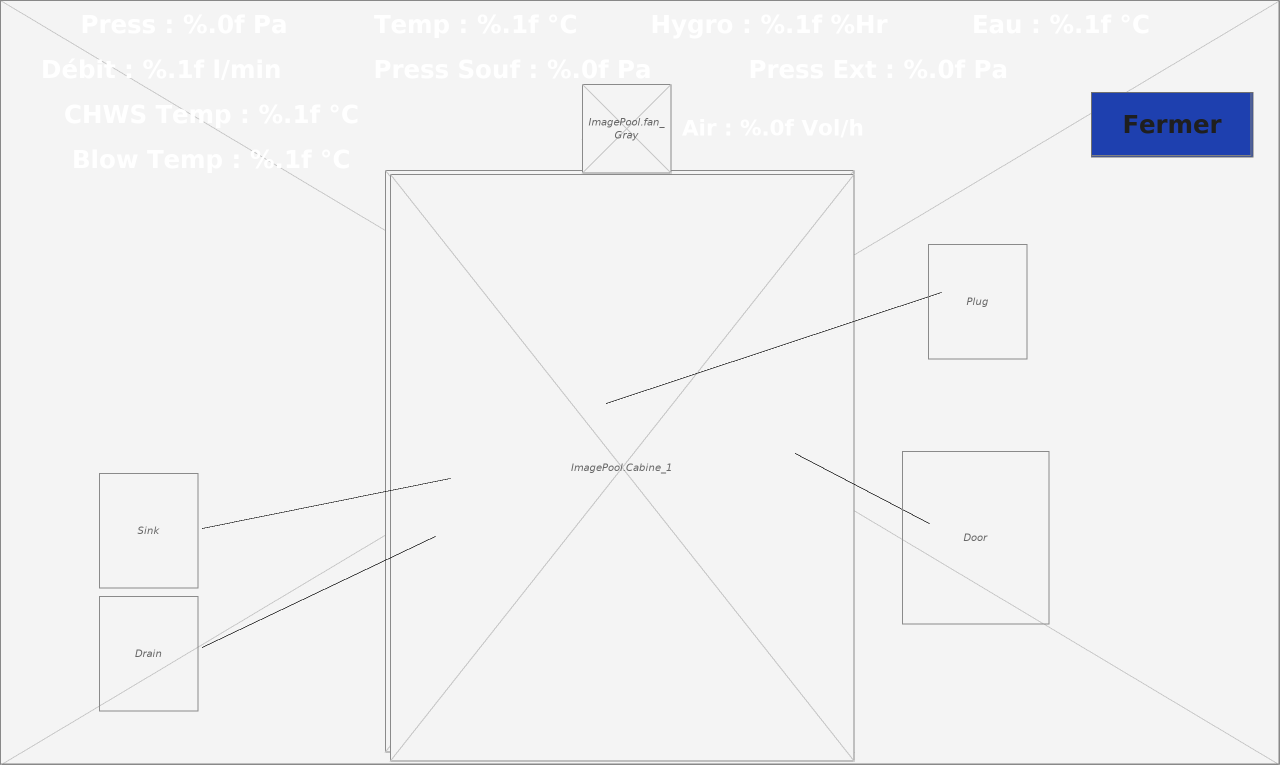
VISUALIZATION Actionneurs  // 1280x765
    Image (0,0 1280x765), image: ImagePool.Fond_Degr
    Image (385,170 469x582), image: ImagePool.Cabine-2
    Polygon (412,662) (553,704) (695,739) (769,704) (844,662), colour variable: GVL_Visu.Couleur_Cabine
    Polygon (414,662) (412,248) (697,187) (840,256) (842,662), colour variable: GVL_Visu.Couleur_Cabine
    Image (390,174 464x587), image: ImagePool.Cabine_1
    Line (202,528) (450,478)
    Line (795,453) (929,523)
    Line (606,403) (941,292)
    Button (1091,92 162x65), "Fermer"
        OnMouseDown: CloseDialog Dialog=Actionneurs, Result=OK, NumpadKeypadSet=True
    Group (582,84 393x89), invisible if: TRUE
        Rectangle (97,23 296x42), "Air : %.0f Vol/h", text variable: MES_Debit_Volh_Soufflage
        Group (0,0 89x89), invisible if: NOT Visu.On_Off_Ventilation
            Image (0,0 55x55), invisible if: NOT GVL_Visu.On_Off_Anim, image: ImagePool.fan_45
            Image (0,0 55x55), invisible if: GVL_Visu.On_Off_Anim, image: ImagePool.fan (1)
        Image (0,0 89x89), invisible if: Visu.On_Off_Ventilation, image: ImagePool.fan_Gray
    Frame (99,473 99x115)
        shows Sink(Etat_MaAr := S_Cmd_ElectroValve_Alim_Lavabo)
    Line (202,647) (435,536)
    Frame (902,451 147x173)
        shows Door(Etat_MaAr := E_Info_Contact_Porte)
    Frame (928,244 99x115)
        shows Plug(Etat_MaAr := S_Cmd_PC_Cab)
    Frame (99,596 99x115)
        shows Drain(Etat_MaAr := S_Cmd_Vanne_Vid_Lavabo)
    Rectangle (623,2 292x45), "Hygro : %.1f %Hr", text variable: Tab_MES_Sonde_Hygro_Amb.R_MesCor
    Rectangle (330,2 292x45), "Temp : %.1f °C", text variable: Tab_MES_Sonde_Temp_Amb.R_MesCor
    Rectangle (38,2 292x45), "Press : %.0f Pa", text variable: Tab_MES_Sonde_Press_Cab.R_MesCor
    Rectangle (915,2 292x45), "Eau : %.1f °C", text variable: MES_Temp_Eau_Mitige_General
    Rectangle (38,47 292x45), "Débit : %.1f l/min", text variable: GVL_Visu.Visu_Mes_Debit_Eau_Manu, invisible if: NOT a5_Ecriture_InterCom.Dmd_Mise_En_Temp
    Rectangle (330,47 365x45), "Press Souf : %.0f Pa", text variable: Tab_Mes_Sonde_Pression_Souf.R_MesCor, invisible if: NOT Option_Press_SoufExt_General
    Rectangle (696,47 365x45), "Press Ext : %.0f Pa", text variable: Tab_Mes_Sonde_Pression_Ext.R_MesCor, invisible if: NOT Option_Press_SoufExt_General
    Rectangle (38,92 347x45), "CHWS Temp : %.1f °C", text variable: Tab_Mes_Sonde_Temp_BatEG.R_MesCor
    Rectangle (38,137 347x45), "Blow Temp : %.1f °C", text variable: Tab_Mes_Sonde_Temp_Souf.R_MesCor
END_VISUALIZATION

(* stored: Version 1.1.0.1, ProductVersion 3.1.4024.16
   Visu Actionneurs: Id {5f77ef2b-8df6-4a20-9965-009b6cf5b2b1} *)
